FUNCTION FC_Conversion : REAL
VAR_INPUT
	I4 		: 	INT;
	Vmin 	: 	REAL;
	Vmax 	:	REAL;
END_VAR
	
VAR
	Rin	: REAL;
END_VAR

VAR CONSTANT
	Livelli	:	REAL	:= 	32767.0;
END_VAR

Rin	:= INT_TO_REAL(I4);
FC_Conversion	:=	Rin/Livelli*(Vmax-Vmin)/2.0;

END_FUNCTION

(* stored: Version 1.1.0.1, ProductVersion 3.1.4024.12
   POU FC_Conversion: Id {71233210-eb77-456c-89ed-7fd6401d34bc}, SpecialFunc None *)
